(*********************************** G.D S.p.A. - Technical Department ***********************************
============= PROGRAM INFO ============
FOLDER:             TBD
MACHINES INVOLVED:  TBD 

============= DESCRIPTION =============
csp machine declaration

============= REVISIONS ===============
Date		Version	 	Author      	Description             
----------	-------		------------  	--------------------------------------------
2019/04/05 	0000.00	 	M.Grasso		Creation of the PRG

**********************************************************************************************************)
(*$R process_ref := prc; $*)
PROGRAM csp_case_discharge
VAR
		
	prc:											process;
	prc_path:										STRING;
	
END_VAR

_read_var_input();

_object_manager();

IF NOT objects_running()
THEN
	RETURN;	
END_IF

_read_process_image();

_mode_manager();

_set_runtime_properties();

(********************************* BODY *********************************)
(************************************************************************)

_handle_messages();

_write_output();

ACTION _handle_messages:
;
END_ACTION

ACTION _handle_process_test:
;
END_ACTION

ACTION _mode_manager:
IF process_mode_req_is_pending(prc)
THEN
    process_apply_mode_req_first_step(prc);
    CASE process_get_mode(prc) OF
        MODE_TO_ABSENT:
			;
        MODE_TO_INACTIVE:
			;
        MODE_TO_TEST:
			;
        MODE_TO_OPERATIONAL:
			;
    END_CASE
    process_apply_mode_req_second_step(prc);
END_IF
END_ACTION

ACTION _object_manager:
IF objects_initialization()
THEN
	sub_process_init(
		object_name					:= 'csp_case_discharge.prc', 
		process						:= csp_case.prc, 
		CONVERSION_this				:= prc);
		
	prc_path 						:= process_get_path(prc);
END_IF

IF objects_running()
THEN
	process_cycle(prc);
END_IF
END_ACTION

ACTION _read_process_image:
;
END_ACTION

ACTION _read_var_input:
;
END_ACTION

ACTION _set_runtime_properties:
;
END_ACTION

ACTION _write_output:
;
END_ACTION

END_PROGRAM

(* stored: Version 1.1.0.1, ProductVersion 3.1.4024.3
   POU csp_case_discharge: Id {562fae22-ddff-4172-94f1-4980bc28b962}, SpecialFunc None
   Action _handle_messages: Id {af1deb5b-680c-4b99-8428-18e170391ff3}
   Action _handle_process_test: Id {ffaff9dc-6f94-42ec-ba10-c51bceaafd5e}
   Action _mode_manager: Id {e9ce68af-34c7-41dc-aa58-284a76e86560}
   Action _object_manager: Id {b8cf93b6-1721-4580-9086-53750b2b6bfe}
   Action _read_process_image: Id {9c81092e-9d1c-4200-b99f-a8c6602aec5c}
   Action _read_var_input: Id {df3d58e9-27df-456b-9ccd-fe95512a7ae8}
   Action _set_runtime_properties: Id {c323d002-fab6-4700-b659-015d0d9c9ec9}
   Action _write_output: Id {7dc0c23d-a2af-4993-bbd8-30f3ddbb456c} *)
